TYPE WARMStruct :
STRUCT
	showText		:STRING:='********';// 提示内容
	showFlag		:BOOL;// 提示显示
	btTrig			:BOOL;// 触发按钮			
	bOK				:BOOL;
	bNO				:BOOL;
END_STRUCT
END_TYPE

(* stored: Version 1.1.0.1, ProductVersion 3.1.4024.4
   DUT WARMStruct: Id {ea6c03b3-b680-4749-a11b-d0ec26528f7a} *)
